# EPICS substitutions: COORD/COORD-IOC-01App/db/riken_port_changeover_groups.substitutions
file riken_port_changeover_groups.template {

pattern {P, GRP}
    {"\$(P)", "1"}
    {"\$(P)", "2"}
    {"\$(P)", "3"}
    {"\$(P)", "4"}
}
